PROGRAM MAIN
VAR
	
	tPulse AT %I*: T_DCTIME64;
	tPrev : T_DCTIME64;
	tPrevPulse : T_DCTIME64;
	tDiff : T_DCTIME64;
	
	SyncMaster : AXIS_REF;
	SyncSlave : AXIS_REF;

	XFC_Position : XFC_PositionAtTime;
	
	fPosition : LREAL;
	fPositionMod : LREAL;
	fPrevPosition : LREAL;
	
	fPositionError : LREAL;
	fPositionSum : LREAL;
	
	fSpeedError : LREAL;
	fSpeedAct : LREAL;
	fSpeed : LREAL := 360*14;
	
	fPositionDiff : LREAL;
	
	Master : AxisController;
	Slave : CamInController;
	
	mcMoveVelo : MC_MoveVelocity;
	
	iState : UINT;
	bPulse : BOOL;
	
	fSpeed_Kp : LREAL := 0.1;
	
	fPosition_Kp : LREAL := 0.1;
	fPosition_Ki : LREAL := 0.001;
	
	fPositionControlThreshold: LREAL := 10;
	
END_VAR

Master(Axis:=SyncMaster);
Master.bExecute:=FALSE;

Slave(Axis:=SyncSlave, Master:=SyncMaster);
Slave.bExecute:=FALSE;

mcMoveVelo(Axis:=SyncMaster);
mcMoveVelo.Execute := FALSE;

CASE iState OF
	000:
		// Compose a camming table?
		
		iState := 100;

	100:
		// Set up the master axis
		Master.fSpeed:=0;
		Master.bExecute := TRUE;
		iState := 101;
	101:
		IF Master.bDone THEN
			iState:= 200;
		END_IF
		
	200:
		// Check for new pulse
		IF tPulse <> tPrev THEN
			// There's a new pusle
			fPrevPosition := fPosition;
			tPrevPulse := tPrev;
			bPulse := TRUE;
		
			// Get the position at the pulse
			XFC_Position(DcTime:=ULINT_TO_UDINT(tPulse), Axis:= SyncMaster);
			fPosition := XFC_Position.Position;
			fPositionMod := MODULO(XFC_Position.Position+180, 360)-180;
			
			// Calculate the distance moved
			fPositionDiff := fPosition-fPrevPosition;
			
			// Calculate the time between pulses
			tDiff := tPulse - tPrevPulse;
			
			// Calculate the actual speed
			fSpeedAct := fPositionDiff/tDiff*1E9;
			
			// Calculate the speed difference - with respect to the expected 360degrees
			fSpeedError := -(fPositionDiff-360)/tDiff*1E9;
			
			// Implement the speed PI controller
			fSpeed := fSpeed + fSpeedError*fSpeed_Kp;
			
			// Implement the position PI controller
			fPositionError := MODULO(fPosition+180, 360)-180;
			fPositionSum := fPositionSum + fPositionError;
			
			// Only activate position control if the speed control is good
			IF ABS(fSpeedError) < fPositionControlThreshold THEN
				fSpeed := fSpeed - fPositionError * fPosition_Kp;
				fSpeed := fSpeed - fPositionSum * fPosition_Ki;
			ELSE
				fPositionSum := 0;
			END_IF
			
			IF fSpeed > 5700 THEN
				fSpeed := 5700;
			END_IF
			
			// Update the velocity
			mcMoveVelo.Execute:= TRUE;
			mcMoveVelo.Velocity:= fSpeed;
			
			(*// Activate slave camming?
			IF NOT Slave.bDone THEN
				Slave.bExecute:=TRUE;
			END_IF*)
		
		ELSE
			bPulse := FALSE;
		END_IF
		
		tPrev := tPulse;
			
END_CASE

END_PROGRAM

(* stored: Version 1.1.0.1, ProductVersion 3.1.4022.10
   POU MAIN: Id {a5509ff2-383d-4902-af38-fb16f957d213}, SpecialFunc None *)
